FUNCTION anyToString : MaxString
VAR_INPUT
  toTransform: ANY;
END_VAR
VAR
  intPtr: POINTER TO INT;
  realPtr: POINTER TO REAL;
  stringPtr: POINTER TO STRING;
END_VAR

CASE UDINT_TO_INT(toTransform.TypeClass) OF
TypeClass.TYPE_INT:
  intPtr := toTransform.pValue;
  anyToString := TO_STRING(intPtr^);
TypeClass.TYPE_REAL:
  realPtr := toTransform.pValue;
  anyToString := TO_STRING(realPtr^);
TypeClass.TYPE_STRING:
  stringPtr := toTransform.pValue;
  anyToString := stringPtr^;
ELSE
  anyToString := '';
END_CASE

END_FUNCTION

(* stored: Version 1.1.0.1, ProductVersion 3.1.4022.12
   POU anyToString: Id {ac8c30cd-67ee-4e25-b911-ae2d14e6a975}, SpecialFunc None *)
